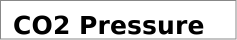
VISUALIZATION VISU_HMI_CO2_PRESSURE  // 237x40
    Label (10,10 227x30), "CO2 Pressure"
END_VISUALIZATION

(* stored: Version 1.1.0.1, ProductVersion 3.1.4024.14
   Visu VISU_HMI_CO2_PRESSURE: Id {cb8d81ab-d66c-4e79-bfc5-f811b8e25e8e} *)
